FUNCTION_BLOCK ObserveStack EXTENDS HardwareObservationBase
VAR_INPUT
END_VAR
VAR_OUTPUT
END_VAR
VAR
	m_ptrStack: POINTER TO Stack;
	m_ptrStackWP: POINTER TO xPPUProduct;
	
	m_rtPresent: R_TRIG;
	m_rtLight: R_TRIG;
	m_rtMetal: R_TRIG;
END_VAR

METHOD FB_init : BOOL
VAR_INPUT
	bInitRetains : BOOL; // if TRUE, the retain variables are initialized (warm start / cold start)
	bInCopyCode : BOOL;  // if TRUE, the instance afterwards gets moved into the copy code (online change)

	i_ptrStack: POINTER TO Stack;
	i_ptrWP: POINTER TO IProduct;
END_VAR
m_ptrStack := i_ptrStack;
IF NOT __QUERYPOINTER(i_ptrWP^, m_ptrStackWP) THEN
	FB_init := FALSE;
END_IF
END_METHOD

METHOD  ResetDefinition : BOOL
VAR_INPUT
END_VAR
;
END_METHOD

(* Update an instance of ProcessState with the part of the process that can be observed by this Hardware Interface. *)
METHOD UpdateProcessObservation : BOOL
VAR_IN_OUT
	io_processState: ProcessState;
END_VAR
io_processState.UpdateState_Binary(EProcessVariables.Stack_WorkpieceAvailable, m_ptrStack^.WPOnTray, i_force := TRUE);

io_processState.UpdateState_Defined(EProcessVariables.Stack_WorkpieceAvailable, TRUE);

// update WP info (if there are sensors available), then update the process variables list
m_rtPresent(CLK := m_ptrStack^.WPOnTray);
m_rtLight(CLK := m_ptrStack^.LightWPOnTray);
m_rtMetal(CLK := m_ptrStack^.MetalWPOnTray);
IF m_rtPresent.Q THEN
	m_ptrStackWP^.IsPresent := TRUE;
END_IF
IF m_rtLight.Q THEN
	m_ptrStackWP^.IsLight := TRUE;
END_IF
IF m_rtMetal.Q THEN
	m_ptrStackWP^.IsMetal := TRUE;
END_IF
io_processState.UpdateState_Numeric(EProcessVariables.Stack_ProductType, UINT_TO_LREAL(m_ptrStackWP^.Material), TRUE);
io_processState.UpdateState_Defined(EProcessVariables.Stack_ProductType, TRUE);
END_METHOD

END_FUNCTION_BLOCK

(* stored: Version 1.1.0.1, ProductVersion 3.1.4024.12
   POU ObserveStack: Id {486ad608-7670-4a46-be68-3129ff7847f4}, SpecialFunc None
   Method FB_init: Id {3c4742fa-36b2-4b1d-9138-ddf77a52c251}
   Method ResetDefinition: Id {9f74f777-c0b1-491e-bfee-41628a59ea39}
   Method UpdateProcessObservation: Id {7817ad32-9b15-4a55-ba2c-9bdf7f27bd75} *)
